# B&R Automation Studio project CleanChemi_SiteManagementSystem (part 24)

```iecst
		IF gSkid_LR[IdxSkids_LR].Alarms.ALARM_P203.11 AND gServices.Alarms.Internal.Alarms_State_LR[IdxSkids_LR].ALARM_P203.11 = FALSE THEN
			IF gSkid_LR[IdxSkids_LR].ErrorInfo.Text = '' THEN
				gSkid_LR[IdxSkids_LR].ErrorInfo.Text		:= 'ALARM_P203.11';
				gSkid_LR[IdxSkids_LR].ErrorInfo.State		:= 'Warning';
				gSkid_LR[IdxSkids_LR].ErrorInfo.Severity	:= 2;
				gSkid_LR[IdxSkids_LR].Error := TRUE;
				gServices.Alarms.Internal.Alarms_State_LR[IdxSkids_LR].ALARM_P203.11 := TRUE;
			END_IF
		END_IF;

		IF gSkid_LR[IdxSkids_LR].Alarms.ALARM_P203.12 AND gServices.Alarms.Internal.Alarms_State_LR[IdxSkids_LR].ALARM_P203.12 = FALSE THEN
			IF gSkid_LR[IdxSkids_LR].ErrorInfo.Text = '' THEN
				gSkid_LR[IdxSkids_LR].ErrorInfo.Text		:= 'ALARM_P203.12';
				gSkid_LR[IdxSkids_LR].ErrorInfo.State		:= 'Warning';
				gSkid_LR[IdxSkids_LR].ErrorInfo.Severity	:= 2;
				gSkid_LR[IdxSkids_LR].Error := TRUE;
				gServices.Alarms.Internal.Alarms_State_LR[IdxSkids_LR].ALARM_P203.12 := TRUE;
			END_IF
		END_IF;

		IF gSkid_LR[IdxSkids_LR].Alarms.ALARM_P203.13 AND gServices.Alarms.Internal.Alarms_State_LR[IdxSkids_LR].ALARM_P203.13 = FALSE THEN
			IF gSkid_LR[IdxSkids_LR].ErrorInfo.Text = '' THEN
				gSkid_LR[IdxSkids_LR].ErrorInfo.Text		:= 'ALARM_P203.13';
				gSkid_LR[IdxSkids_LR].ErrorInfo.State		:= 'Warning';
				gSkid_LR[IdxSkids_LR].ErrorInfo.Severity	:= 2;
				gSkid_LR[IdxSkids_LR].Error := TRUE;
				gServices.Alarms.Internal.Alarms_State_LR[IdxSkids_LR].ALARM_P203.13 := TRUE;
			END_IF
		END_IF;

		IF gSkid_LR[IdxSkids_LR].Alarms.ALARM_P203.14 AND gServices.Alarms.Internal.Alarms_State_LR[IdxSkids_LR].ALARM_P203.14 = FALSE THEN
			IF gSkid_LR[IdxSkids_LR].ErrorInfo.Text = '' THEN
				gSkid_LR[IdxSkids_LR].ErrorInfo.Text		:= 'ALARM_P203.14';
				gSkid_LR[IdxSkids_LR].ErrorInfo.State		:= 'Warning';
				gSkid_LR[IdxSkids_LR].ErrorInfo.Severity	:= 2;
				gSkid_LR[IdxSkids_LR].Error := TRUE;
				gServices.Alarms.Internal.Alarms_State_LR[IdxSkids_LR].ALARM_P203.14 := TRUE;
			END_IF
		END_IF;

		IF gSkid_LR[IdxSkids_LR].Alarms.ALARM_P203.15 AND gServices.Alarms.Internal.Alarms_State_LR[IdxSkids_LR].ALARM_P203.15 = FALSE THEN
			IF gSkid_LR[IdxSkids_LR].ErrorInfo.Text = '' THEN
				gSkid_LR[IdxSkids_LR].ErrorInfo.Text		:= 'ALARM_P203.15';
				gSkid_LR[IdxSkids_LR].ErrorInfo.State		:= 'Warning';
				gSkid_LR[IdxSkids_LR].ErrorInfo.Severity	:= 2;
				gSkid_LR[IdxSkids_LR].Error := TRUE;
				gServices.Alarms.Internal.Alarms_State_LR[IdxSkids_LR].ALARM_P203.15 := TRUE;
			END_IF
		END_IF;
	END_IF;

	(*********************************************************************Dont Touch This Code**********************************************************************)
	IF gSkid_LR[IdxSkids_LR].Error AND gSkid_LR[IdxSkids_LR].AlarmsInitialized AND gSkid_LR[IdxSkids_LR].Pmax_General_Variables.UNIT_ID <> 0 AND gUnit_LR[IdxSkids_LR] <> 0 THEN
		CASE gSkid_LR[IdxSkids_LR].ErrorInfo.Severity OF
			1:
				gSkid_LR[IdxSkids_LR].tempAlarm.name				:= UINT_TO_STRING(gUnit_LR[IdxSkids_LR]);
				gSkid_LR[IdxSkids_LR].tempAlarm.name				:= CONCAT('Skid',gSkid_LR[IdxSkids_LR].tempAlarm.name);
				gSkid_LR[IdxSkids_LR].tempAlarm.name				:= CONCAT(gSkid_LR[IdxSkids_LR].tempAlarm.name,'Severity1');
				gSkid_LR[IdxSkids_LR].tempAlarm.allowMultiple		:= TRUE;
				gSkid_LR[IdxSkids_LR].tempAlarm.addText[0]		:= gSkid_LR[IdxSkids_LR].ErrorInfo.State;
				gSkid_LR[IdxSkids_LR].tempAlarm.addText[1]		:= gSkid_LR[IdxSkids_LR].ErrorInfo.Text;

				HA_Array_AddTop(ADR(gServices.Alarms.In.AlarmList), SIZEOF(gServices.Alarms.In.AlarmList), ADR(gSkid_LR[IdxSkids_LR].tempAlarm), SIZEOF(gSkid_LR[IdxSkids_LR].tempAlarm));
			2:
				gSkid_LR[IdxSkids_LR].tempAlarm.name				:=  UINT_TO_STRING(gUnit_LR[IdxSkids_LR]);
				gSkid_LR[IdxSkids_LR].tempAlarm.name				:= CONCAT('Skid',gSkid_LR[IdxSkids_LR].tempAlarm.name);
				gSkid_LR[IdxSkids_LR].tempAlarm.name				:= CONCAT(gSkid_LR[IdxSkids_LR].tempAlarm.name,'Severity2');
				gSkid_LR[IdxSkids_LR].tempAlarm.allowMultiple		:= TRUE;
				gSkid_LR[IdxSkids_LR].tempAlarm.addText[0]		:= gSkid_LR[IdxSkids_LR].ErrorInfo.State;
				gSkid_LR[IdxSkids_LR].tempAlarm.addText[1]		:= gSkid_LR[IdxSkids_LR].ErrorInfo.Text;

				HA_Array_AddTop(ADR(gServices.Alarms.In.AlarmList), SIZEOF(gServices.Alarms.In.AlarmList), ADR(gSkid_LR[IdxSkids_LR].tempAlarm), SIZEOF(gSkid_LR[IdxSkids_LR].tempAlarm));
			3:
				gSkid_LR[IdxSkids_LR].tempAlarm.name				:=  UINT_TO_STRING(gUnit_LR[IdxSkids_LR]);
				gSkid_LR[IdxSkids_LR].tempAlarm.name				:= CONCAT('Skid',gSkid_LR[IdxSkids_LR].tempAlarm.name);
				gSkid_LR[IdxSkids_LR].tempAlarm.name				:= CONCAT(gSkid_LR[IdxSkids_LR].tempAlarm.name,'Severity3');
				gSkid_LR[IdxSkids_LR].tempAlarm.allowMultiple		:= TRUE;
				gSkid_LR[IdxSkids_LR].tempAlarm.addText[0]		:= gSkid_LR[IdxSkids_LR].ErrorInfo.State;
				gSkid_LR[IdxSkids_LR].tempAlarm.addText[1]		:= gSkid_LR[IdxSkids_LR].ErrorInfo.Text;

				HA_Array_AddTop(ADR(gServices.Alarms.In.AlarmList), SIZEOF(gServices.Alarms.In.AlarmList), ADR(gSkid_LR[IdxSkids_LR].tempAlarm), SIZEOF(gSkid_LR[IdxSkids_LR].tempAlarm));
			4:
				gSkid_LR[IdxSkids_LR].tempAlarm.name				:=  UINT_TO_STRING(gUnit_LR[IdxSkids_LR]);
				gSkid_LR[IdxSkids_LR].tempAlarm.name				:= CONCAT('Skid',gSkid_LR[IdxSkids_LR].tempAlarm.name);
				gSkid_LR[IdxSkids_LR].tempAlarm.name				:= CONCAT(gSkid_LR[IdxSkids_LR].tempAlarm.name,'Severity4');
				gSkid_LR[IdxSkids_LR].tempAlarm.allowMultiple		:= TRUE;
				gSkid_LR[IdxSkids_LR].tempAlarm.addText[0]		:= gSkid_LR[IdxSkids_LR].ErrorInfo.State;
				gSkid_LR[IdxSkids_LR].tempAlarm.addText[1]		:= gSkid_LR[IdxSkids_LR].ErrorInfo.Text;

				HA_Array_AddTop(ADR(gServices.Alarms.In.AlarmList), SIZEOF(gServices.Alarms.In.AlarmList), ADR(gSkid_LR[IdxSkids_LR].tempAlarm), SIZEOF(gSkid_LR[IdxSkids_LR].tempAlarm));
			5:

				gSkid_LR[IdxSkids_LR].tempAlarm.name				:=  UINT_TO_STRING(gUnit_LR[IdxSkids_LR]);
				gSkid_LR[IdxSkids_LR].tempAlarm.name				:= CONCAT('Skid',gSkid_LR[IdxSkids_LR].tempAlarm.name);
				gSkid_LR[IdxSkids_LR].tempAlarm.name				:= CONCAT(gSkid_LR[IdxSkids_LR].tempAlarm.name,'Severity5');
				gSkid_LR[IdxSkids_LR].tempAlarm.allowMultiple		:= TRUE;
				gSkid_LR[IdxSkids_LR].tempAlarm.addText[0]		:= gSkid_LR[IdxSkids_LR].ErrorInfo.State;
				gSkid_LR[IdxSkids_LR].tempAlarm.addText[1]		:= gSkid_LR[IdxSkids_LR].ErrorInfo.Text;

				HA_Array_AddTop(ADR(gServices.Alarms.In.AlarmList), SIZEOF(gServices.Alarms.In.AlarmList), ADR(gSkid_LR[IdxSkids_LR].tempAlarm), SIZEOF(gSkid_LR[IdxSkids_LR].tempAlarm));
		END_CASE

		gSkid_LR[IdxSkids_LR].Error := FALSE;

	END_IF

	brsmemset(ADR(gSkid_LR[IdxSkids_LR].ErrorInfo),0,SIZEOF(gSkid_LR[IdxSkids_LR].ErrorInfo));

	gServices.Alarms.Internal.MpAlarmXHistory_0.DeviceName 						:= ADR(gServices.DeviceName);

	//Set Unit Number and Add Alarms
	IF (gSkid_LR[IdxSkids_LR].Pmax_General_Variables.UNIT_ID <> 0 AND (gUnit_LR[IdxSkids_LR] <> gSkid_LR[IdxSkids_LR].Pmax_General_Variables.UNIT_ID))
		OR (gUnit_LR[IdxSkids_LR] <> 0 AND gVis.Alarms.Active.FilterString_LR[IdxSkids_LR] = '') THEN

		gUnit_LR[IdxSkids_LR] := gSkid_LR[IdxSkids_LR].Pmax_General_Variables.UNIT_ID;

		gSkid_LR[IdxSkids_LR].AlarmName	 := UINT_TO_STRING(gUnit_LR[IdxSkids_LR]);
		gSkid_LR[IdxSkids_LR].AlarmName	 := CONCAT('Skid',gSkid_LR[IdxSkids_LR].AlarmName	);

		gSkid_LR[IdxSkids_LR].i := 1;

		SkidNumberINT := UINT_TO_STRING(gUnit_LR[IdxSkids_LR]);

		gVis.Alarms.Active.FilterString_LR[IdxSkids_LR] := CONCAT('[{"value":',SkidNumberINT);
		gVis.Alarms.Active.FilterString_LR[IdxSkids_LR] :=  CONCAT(gVis.Alarms.Active.FilterString_LR[IdxSkids_LR] ,',"conditionType":"==","columnPosition":1}]');

	END_IF;

	// Case for handling the alarm history
	CASE gServices.Alarms.Internal.StateExportHistory OF
		0:
			IF gServices.Alarms.In.ExportHistory THEN
				HA_AlarmX_Helper(gAlarmXCore,'',HA_ALARMX_ACTION_LOG_ONLY,'HISTORY EXPORTED',FALSE);
				gServices.Alarms.In.ExportHistory 									:= FALSE;
				gServices.Alarms.Internal.MpAlarmXHistory_0.Export 				:= TRUE;
				gServices.Alarms.Internal.StateExportHistory 						:= 10;
			ELSIF gServices.Alarms.In.ClearHistory THEN
				HA_AlarmX_Helper(gAlarmXCore,'',HA_ALARMX_ACTION_LOG_ONLY,'HISTORY CLEARED',FALSE);
				gServices.Alarms.In.ClearHistory 									:= FALSE;
				MpAlarmXClearHistory(gAlarmXHistory);
			END_IF;
		10:
			IF gServices.Alarms.Internal.MpAlarmXHistory_0.CommandDone OR gServices.Alarms.Internal.MpAlarmXHistory_0.Error THEN
				gServices.Alarms.Internal.MpAlarmXHistory_0.Export 				:= FALSE;
				gServices.Alarms.Internal.StateExportHistory 						:= 0;
			END_IF;
	END_CASE;

	//	IF gMain.ErrorReset THEN
	//		gServices.Alarms.In.ResetAlarms 											:= TRUE;
	//	END_IF;

	// Case for handling the alarm resetting
	CASE gServices.Alarms.Internal.StateResetAlarms OF
		0:
			IF gServices.Alarms.In.ResetAlarms OR gVis.Global.ErrorReset THEN
				HA_AlarmX_Helper(gAlarmXCore,'',HA_ALARMX_ACTION_LOG_ONLY,'ACKNOWLEDGE ALL',FALSE);
				gServices.Alarms.In.ResetAlarms 									:= FALSE;
				gVis.Alarms.Active.UIConnect.AcknowledgeAll 							:= TRUE;
				gServices.Alarms.Internal.CTON_ResetDelay(IN := FALSE);
				gServices.Alarms.Internal.StateResetAlarms 						:= 10;
			END_IF;
		10:
			// give UI time to process the reset
			IF gServices.Alarms.Internal.CTON_ResetDelay.Q THEN
				gServices.Alarms.Internal.CTON_ResetDelay(IN := FALSE);
				gServices.Alarms.Internal.StateResetAlarms 						:= 0;
				gVis.Global.ErrorReset := FALSE;
			ELSE
				gServices.Alarms.Internal.CTON_ResetDelay(IN := TRUE, PT := T#250ms);
			END_IF;
	END_CASE;

	//Create Alarms
	CASE gSkid_LR[IdxSkids_LR].i OF
		0:
			//IDLE
		1:
			gSkid_LR[IdxSkids_LR].AlarmName	 := UINT_TO_STRING(gUnit_LR[IdxSkids_LR]);
			gSkid_LR[IdxSkids_LR].AlarmName	 := CONCAT('Skid',gSkid_LR[IdxSkids_LR].AlarmName	);
			HA_brsstrcat(ADR(gSkid_LR[IdxSkids_LR].AlarmName), ADR('Severity1'), SIZEOF(gSkid_LR[IdxSkids_LR].AlarmName));
			gSkid_LR[IdxSkids_LR].AlarmCfg.Message												:= '{$$IAT/Alarm.';
			HA_brsstrcat(ADR(gSkid_LR[IdxSkids_LR].AlarmCfg.Message), ADR('Severity1'), SIZEOF(gSkid_LR[IdxSkids_LR].AlarmCfg.Message));
			HA_brsstrcat(ADR(gSkid_LR[IdxSkids_LR].AlarmCfg.Message), ADR('}'), SIZEOF(gSkid_LR[IdxSkids_LR].AlarmCfg.Message));
			gSkid_LR[IdxSkids_LR].AlarmCfg.Code													:= gUnit_LR[IdxSkids_LR];
			gSkid_LR[IdxSkids_LR].AlarmCfg.Severity												:= 1;
			gSkid_LR[IdxSkids_LR].AlarmCfg.Behavior.AutoReset									:= TRUE;
			gSkid_LR[IdxSkids_LR].AlarmCfg.Behavior.Acknowledge 									:= mpALARMX_ACK_REQ;
			gSkid_LR[IdxSkids_LR].AlarmCfg.Behavior.MultipleInstances 							:= TRUE;
			gSkid_LR[IdxSkids_LR].AlarmCfg.Behavior.ReactionUntilAcknowledged					:= TRUE;
			gSkid_LR[IdxSkids_LR].AlarmCfg.Behavior.HistoryReport.AcknowledgedToUnacknowledged := FALSE;
			gSkid_LR[IdxSkids_LR].AlarmCfg.Behavior.HistoryReport.ActiveToInactive := FALSE;
			gSkid_LR[IdxSkids_LR].AlarmCfg.Behavior.HistoryReport.InactiveToActive := TRUE;
			gSkid_LR[IdxSkids_LR].AlarmCfg.Behavior.HistoryReport.Reactivation := FALSE;
			gSkid_LR[IdxSkids_LR].AlarmCfg.Behavior.HistoryReport.UnacknowledgedToAcknowledged := FALSE;
			gSkid_LR[IdxSkids_LR].MpAlarmXConfigAlarm.Save				:= TRUE;

		2:
			gSkid_LR[IdxSkids_LR].AlarmName	 := UINT_TO_STRING(gUnit_LR[IdxSkids_LR]);
			gSkid_LR[IdxSkids_LR].AlarmName	 := CONCAT('Skid',gSkid_LR[IdxSkids_LR].AlarmName	);
			HA_brsstrcat(ADR(gSkid_LR[IdxSkids_LR].AlarmName), ADR('Severity2'), SIZEOF(gSkid_LR[IdxSkids_LR].AlarmName));
			gSkid_LR[IdxSkids_LR].AlarmCfg.Message												:= '{$$IAT/Alarm.';
			HA_brsstrcat(ADR(gSkid_LR[IdxSkids_LR].AlarmCfg.Message), ADR('Severity2'), SIZEOF(gSkid_LR[IdxSkids_LR].AlarmCfg.Message));
			HA_brsstrcat(ADR(gSkid_LR[IdxSkids_LR].AlarmCfg.Message), ADR('}'), SIZEOF(gSkid_LR[IdxSkids_LR].AlarmCfg.Message));
			gSkid_LR[IdxSkids_LR].AlarmCfg.Code													:= gUnit_LR[IdxSkids_LR];
			gSkid_LR[IdxSkids_LR].AlarmCfg.Severity												:= 2;
			gSkid_LR[IdxSkids_LR].AlarmCfg.Behavior.AutoReset									:= TRUE;
			gSkid_LR[IdxSkids_LR].AlarmCfg.Behavior.Acknowledge 									:= mpALARMX_ACK_REQ;
			gSkid_LR[IdxSkids_LR].AlarmCfg.Behavior.MultipleInstances 							:= TRUE;
			gSkid_LR[IdxSkids_LR].AlarmCfg.Behavior.ReactionUntilAcknowledged					:= TRUE;
			gSkid_LR[IdxSkids_LR].AlarmCfg.Behavior.HistoryReport.AcknowledgedToUnacknowledged := FALSE;
			gSkid_LR[IdxSkids_LR].AlarmCfg.Behavior.HistoryReport.ActiveToInactive := FALSE;
			gSkid_LR[IdxSkids_LR].AlarmCfg.Behavior.HistoryReport.InactiveToActive := TRUE;
			gSkid_LR[IdxSkids_LR].AlarmCfg.Behavior.HistoryReport.Reactivation := FALSE;
			gSkid_LR[IdxSkids_LR].AlarmCfg.Behavior.HistoryReport.UnacknowledgedToAcknowledged := FALSE;
			gSkid_LR[IdxSkids_LR].MpAlarmXConfigAlarm.Save				:= TRUE;

		3:
			gSkid_LR[IdxSkids_LR].AlarmName	 := UINT_TO_STRING(gUnit_LR[IdxSkids_LR]);
			gSkid_LR[IdxSkids_LR].AlarmName	 := CONCAT('Skid',gSkid_LR[IdxSkids_LR].AlarmName	);
			HA_brsstrcat(ADR(gSkid_LR[IdxSkids_LR].AlarmName), ADR('Severity3'), SIZEOF(gSkid_LR[IdxSkids_LR].AlarmName));
			gSkid_LR[IdxSkids_LR].AlarmCfg.Message												:= '{$$IAT/Alarm.';
			HA_brsstrcat(ADR(gSkid_LR[IdxSkids_LR].AlarmCfg.Message), ADR('Severity3'), SIZEOF(gSkid_LR[IdxSkids_LR].AlarmCfg.Message));
			HA_brsstrcat(ADR(gSkid_LR[IdxSkids_LR].AlarmCfg.Message), ADR('}'), SIZEOF(gSkid_LR[IdxSkids_LR].AlarmCfg.Message));
			gSkid_LR[IdxSkids_LR].AlarmCfg.Code													:= gUnit_LR[IdxSkids_LR];
			gSkid_LR[IdxSkids_LR].AlarmCfg.Severity												:= 3;
			gSkid_LR[IdxSkids_LR].AlarmCfg.Behavior.AutoReset									:= TRUE;
			gSkid_LR[IdxSkids_LR].AlarmCfg.Behavior.Acknowledge 									:= mpALARMX_ACK_REQ;
			gSkid_LR[IdxSkids_LR].AlarmCfg.Behavior.MultipleInstances 							:= TRUE;
			gSkid_LR[IdxSkids_LR].AlarmCfg.Behavior.ReactionUntilAcknowledged					:= TRUE;
			gSkid_LR[IdxSkids_LR].AlarmCfg.Behavior.HistoryReport.AcknowledgedToUnacknowledged := FALSE;
			gSkid_LR[IdxSkids_LR].AlarmCfg.Behavior.HistoryReport.ActiveToInactive := FALSE;
			gSkid_LR[IdxSkids_LR].AlarmCfg.Behavior.HistoryReport.InactiveToActive := TRUE;
			gSkid_LR[IdxSkids_LR].AlarmCfg.Behavior.HistoryReport.Reactivation := FALSE;
			gSkid_LR[IdxSkids_LR].AlarmCfg.Behavior.HistoryReport.UnacknowledgedToAcknowledged := FALSE;
			gSkid_LR[IdxSkids_LR].MpAlarmXConfigAlarm.Save				:= TRUE;

		4:
			gSkid_LR[IdxSkids_LR].AlarmName	 := UINT_TO_STRING(gUnit_LR[IdxSkids_LR]);
			gSkid_LR[IdxSkids_LR].AlarmName	 := CONCAT('Skid',gSkid_LR[IdxSkids_LR].AlarmName	);
			HA_brsstrcat(ADR(gSkid_LR[IdxSkids_LR].AlarmName), ADR('Severity4'), SIZEOF(gSkid_LR[IdxSkids_LR].AlarmName));
			gSkid_LR[IdxSkids_LR].AlarmCfg.Message												:= '{$$IAT/Alarm.';
			HA_brsstrcat(ADR(gSkid_LR[IdxSkids_LR].AlarmCfg.Message), ADR('Severity4'), SIZEOF(gSkid_LR[IdxSkids_LR].AlarmCfg.Message));
			HA_brsstrcat(ADR(gSkid_LR[IdxSkids_LR].AlarmCfg.Message), ADR('}'), SIZEOF(gSkid_LR[IdxSkids_LR].AlarmCfg.Message));
			gSkid_LR[IdxSkids_LR].AlarmCfg.Code													:= gUnit_LR[IdxSkids_LR];
			gSkid_LR[IdxSkids_LR].AlarmCfg.Severity												:= 4;
			gSkid_LR[IdxSkids_LR].AlarmCfg.Behavior.AutoReset									:= TRUE;
			gSkid_LR[IdxSkids_LR].AlarmCfg.Behavior.Acknowledge 									:= mpALARMX_ACK_REQ;
			gSkid_LR[IdxSkids_LR].AlarmCfg.Behavior.MultipleInstances 							:= TRUE;
			gSkid_LR[IdxSkids_LR].AlarmCfg.Behavior.ReactionUntilAcknowledged					:= TRUE;
			gSkid_LR[IdxSkids_LR].AlarmCfg.Behavior.HistoryReport.AcknowledgedToUnacknowledged := FALSE;
			gSkid_LR[IdxSkids_LR].AlarmCfg.Behavior.HistoryReport.ActiveToInactive := FALSE;
			gSkid_LR[IdxSkids_LR].AlarmCfg.Behavior.HistoryReport.InactiveToActive := TRUE;
			gSkid_LR[IdxSkids_LR].AlarmCfg.Behavior.HistoryReport.Reactivation := FALSE;
			gSkid_LR[IdxSkids_LR].AlarmCfg.Behavior.HistoryReport.UnacknowledgedToAcknowledged := FALSE;
			gSkid_LR[IdxSkids_LR].MpAlarmXConfigAlarm.Save				:= TRUE;
		5:
			gSkid_LR[IdxSkids_LR].AlarmName	 := UINT_TO_STRING(gUnit_LR[IdxSkids_LR]);
			gSkid_LR[IdxSkids_LR].AlarmName	 := CONCAT('Skid',gSkid_LR[IdxSkids_LR].AlarmName	);
			HA_brsstrcat(ADR(gSkid_LR[IdxSkids_LR].AlarmName), ADR('Severity5'), SIZEOF(gSkid_LR[IdxSkids_LR].AlarmName));
			gSkid_LR[IdxSkids_LR].AlarmCfg.Message												:= '{$$IAT/Alarm.';
			HA_brsstrcat(ADR(gSkid_LR[IdxSkids_LR].AlarmCfg.Message), ADR('Severity5'), SIZEOF(gSkid_LR[IdxSkids_LR].AlarmCfg.Message));
			HA_brsstrcat(ADR(gSkid_LR[IdxSkids_LR].AlarmCfg.Message), ADR('}'), SIZEOF(gSkid_LR[IdxSkids_LR].AlarmCfg.Message));
			gSkid_LR[IdxSkids_LR].AlarmCfg.Code													:= gUnit_LR[IdxSkids_LR];
			gSkid_LR[IdxSkids_LR].AlarmCfg.Severity												:= 5;
			gSkid_LR[IdxSkids_LR].AlarmCfg.Behavior.AutoReset									:= TRUE;
			gSkid_LR[IdxSkids_LR].AlarmCfg.Behavior.Acknowledge 									:= mpALARMX_ACK_REQ;
			gSkid_LR[IdxSkids_LR].AlarmCfg.Behavior.MultipleInstances 							:= TRUE;
			gSkid_LR[IdxSkids_LR].AlarmCfg.Behavior.ReactionUntilAcknowledged					:= TRUE;
			gSkid_LR[IdxSkids_LR].AlarmCfg.Behavior.HistoryReport.AcknowledgedToUnacknowledged := FALSE;
			gSkid_LR[IdxSkids_LR].AlarmCfg.Behavior.HistoryReport.ActiveToInactive := FALSE;
			gSkid_LR[IdxSkids_LR].AlarmCfg.Behavior.HistoryReport.InactiveToActive := TRUE;
			gSkid_LR[IdxSkids_LR].AlarmCfg.Behavior.HistoryReport.Reactivation := FALSE;
			gSkid_LR[IdxSkids_LR].AlarmCfg.Behavior.HistoryReport.UnacknowledgedToAcknowledged := FALSE;
			gSkid_LR[IdxSkids_LR].MpAlarmXConfigAlarm.Save				:= TRUE;

		6:
			gSkid_LR[IdxSkids_LR].AlarmName	 := UINT_TO_STRING(gUnit_LR[IdxSkids_LR]);
			gSkid_LR[IdxSkids_LR].AlarmName	 := CONCAT('Skid',gSkid_LR[IdxSkids_LR].AlarmName	);
			HA_brsstrcat(ADR(gSkid_LR[IdxSkids_LR].AlarmName), ADR('CmdIgnored'), SIZEOF(gSkid_LR[IdxSkids_LR].AlarmName));
			gSkid_LR[IdxSkids_LR].AlarmCfg.Message												:= '{$$IAT/Alarm.';
			HA_brsstrcat(ADR(gSkid_LR[IdxSkids_LR].AlarmCfg.Message), ADR(gSkid_LR[IdxSkids_LR].AlarmName), SIZEOF(gSkid_LR[IdxSkids_LR].AlarmCfg.Message));
			HA_brsstrcat(ADR(gSkid_LR[IdxSkids_LR].AlarmCfg.Message), ADR('}'), SIZEOF(gSkid_LR[IdxSkids_LR].AlarmCfg.Message));
			gSkid_LR[IdxSkids_LR].AlarmCfg.Code													:= gUnit_LR[IdxSkids_LR] + 6;
			gSkid_LR[IdxSkids_LR].AlarmCfg.Severity												:= 0;
			gSkid_LR[IdxSkids_LR].AlarmCfg.Behavior.AutoReset									:= TRUE;
			gSkid_LR[IdxSkids_LR].AlarmCfg.Behavior.Acknowledge 									:= mpALARMX_ACK_REQ;
			gSkid_LR[IdxSkids_LR].AlarmCfg.Behavior.MultipleInstances 							:= TRUE;
			gSkid_LR[IdxSkids_LR].AlarmCfg.Behavior.ReactionUntilAcknowledged					:= TRUE;
			gSkid_LR[IdxSkids_LR].AlarmCfg.Behavior.HistoryReport.AcknowledgedToUnacknowledged := FALSE;
			gSkid_LR[IdxSkids_LR].AlarmCfg.Behavior.HistoryReport.ActiveToInactive := FALSE;
			gSkid_LR[IdxSkids_LR].AlarmCfg.Behavior.HistoryReport.InactiveToActive := TRUE;
			gSkid_LR[IdxSkids_LR].AlarmCfg.Behavior.HistoryReport.Reactivation := FALSE;
			gSkid_LR[IdxSkids_LR].AlarmCfg.Behavior.HistoryReport.UnacknowledgedToAcknowledged := FALSE;
			gSkid_LR[IdxSkids_LR].MpAlarmXConfigAlarm.Save				:= TRUE;
		7:
			gSkid_LR[IdxSkids_LR].AlarmStartupDelay.IN := TRUE;

			IF 	gSkid_LR[IdxSkids_LR].AlarmStartupDelay.Q THEN
				gSkid_LR[IdxSkids_LR].AlarmsInitialized := TRUE;
			END_IF;

	END_CASE

	gSkid_LR[IdxSkids_LR].AlarmStartupDelay(PT := T#30s);

	gSkid_LR[IdxSkids_LR].MpAlarmXConfigAlarm.MpLink			:= ADR(gAlarmXCore);
	gSkid_LR[IdxSkids_LR].MpAlarmXConfigAlarm.Enable			:= TRUE;
	gSkid_LR[IdxSkids_LR].MpAlarmXConfigAlarm.Name				:= ADR(gSkid_LR[IdxSkids_LR].AlarmName);
	gSkid_LR[IdxSkids_LR].MpAlarmXConfigAlarm.Configuration	:= ADR(gSkid_LR[IdxSkids_LR].AlarmCfg);

	IF gSkid_LR[IdxSkids_LR].MpAlarmXConfigAlarm.CommandDone THEN
		IF gSkid_LR[IdxSkids_LR].i < 7 THEN
			gSkid_LR[IdxSkids_LR].i := gSkid_LR[IdxSkids_LR].i + 1;
		ELSE
			//Do nothing
		END_IF;

		gSkid_LR[IdxSkids_LR].MpAlarmXConfigAlarm.Save := FALSE;
	END_IF;

	gSkid_LR[IdxSkids_LR].MpAlarmXConfigAlarm();

END_ACTION
```

- Visualisation Logical/mappView (not shown)

### Program Logical/Vis (IEC)

#### Main.st - Init, cyclic, exit code
```iecst
PROGRAM _INIT

	brsmemset(ADR(gVis.Main.Out.IPAddressDataProv_HR),0,SIZEOF(gVis.Main.Out.IPAddressDataProv_HR));
	brsmemset(ADR(gVis.Main.Out.IPAddressDataProv_LR),0,SIZEOF(gVis.Main.Out.IPAddressDataProv_LR));

	//Set IP Address for screen
	gVis.Main.Out.SkidIPAddress_LR := SLAVE_IP_ADDRESSES_LR;
	gVis.Main.Out.SkidIPAddress_HR := SLAVE_IP_ADDRESSES_HR;

END_PROGRAM

PROGRAM _CYCLIC

	//Grab Unit ID and Create Dropdown List
	FOR IdxSkids_LR := 0 TO MAX_SKIDS_LR DO

		IF gSkid_LR[IdxSkids_LR].Pmax_General_Variables.UNIT_ID = 0 THEN
			gVis.Main.Internal.IP_WSTRING_Temp := STRING_TO_WSTRING(SLAVE_IP_ADDRESSES_LR[IdxSkids_LR]);
			WString2DataProvider(ADR(gVis.Main.Internal.IP_WSTRING_Temp),IdxSkids_LR,ADR(gVis.Main.Out.IPAddressDataProv_LR[IdxSkids_LR]));
		ELSE
			gVis.Main.Internal.IP_WSTRING_Temp := UINT_TO_WSTRING(gSkid_LR[IdxSkids_LR].Pmax_General_Variables.UNIT_ID );
			WString2DataProvider(ADR(gVis.Main.Internal.IP_WSTRING_Temp),gSkid_LR[IdxSkids_LR].Pmax_General_Variables.UNIT_ID,ADR(gVis.Main.Out.IPAddressDataProv_LR[IdxSkids_LR]));
		END_IF;

	END_FOR

	FOR IdxSkids_HR := 0 TO MAX_SKIDS_HR DO

		IF gSkid_HR[IdxSkids_HR].Pmax_General_Variables.UNIT_ID = 0 THEN
			gVis.Main.Internal.IP_WSTRING_Temp := STRING_TO_WSTRING(SLAVE_IP_ADDRESSES_HR[IdxSkids_HR]);
			WString2DataProvider(ADR(gVis.Main.Internal.IP_WSTRING_Temp),IdxSkids_HR,ADR(gVis.Main.Out.IPAddressDataProv_HR[IdxSkids_HR]));
		ELSE
			gVis.Main.Internal.IP_WSTRING_Temp := UINT_TO_WSTRING(gSkid_HR[IdxSkids_HR].Pmax_General_Variables.UNIT_ID);
			WString2DataProvider(ADR(gVis.Main.Internal.IP_WSTRING_Temp),gSkid_HR[IdxSkids_HR].Pmax_General_Variables.UNIT_ID,ADR(gVis.Main.Out.IPAddressDataProv_HR[IdxSkids_HR]));
		END_IF;

	END_FOR

	//Main Page Widget Vis
	Vis_Main_HR;
	Vis_Main_LR;

	//Vis Action Calls
	Login_User_API;

	//Alarm Page Logic
	Alarms_Active;
	//	Alarms_History;

END_PROGRAM

PROGRAM _EXIT
	(* Insert code here *)

END_PROGRAM
```

#### Types.typ - Local data types
```iecst
TYPE
	USER_LOGIN_ENUM :
		(
		WAITING_FOR_LOGIN_I,
		LOGIN_USER_W,
		LOGIN_USER_C,
		LOGIN_SUCCESS,
		DELETE_USER_C,
		DELETE_USER_W,
		DELETE_USER_SUCCESS,
		DELETE_USER_ERROR,
		LOGIN_ERROR
		);
END_TYPE
```

#### Variables.var - Local variables
```iecst
VAR
	sampleTrigger : BOOL := FALSE;
	samplingTimer : TON := (0);
	bufferIndex : INT := 0;
	SkidNumberINT : STRING[5] := '';
	Idx_AlarmList : INT := 0;
	API_Login_FB_0 : API_Login_FB := (0);
	Header : httpRequestHeader_t := (0);
	CLIENT_LOGIN_STATE : USER_LOGIN_ENUM := WAITING_FOR_LOGIN_I;
	Client : httpsClient := (0);
	IdxClients_AlarmCheck : INT := 0;
	IdxClients : INT := 0;
	ArUserDelete_0 : ArUserDelete := (0);
	ArUserCreate_0 : ArUserCreate := (0);
	IdxSkids_HR : INT := 0;
	IdxSkids_LR : INT := 0;
	IndxNumber : USINT;
END_VAR
```

#### Alarms_Active.st
```iecst
ACTION Alarms_Active:

//	IF gVis.Alarms_Global.Active.Reset THEN
//		gVis.Alarms_Global.Active.Reset											:= FALSE;
//		gVis.Global.ErrorReset													:= TRUE;
//		brsmemset(ADR(gServices.Alarms_Global.Internal.Alarms_State),0,SIZEOF(gServices.Alarms_Global.Internal.Alarms_State));
//	END_IF;
//
	IF gVis.Alarms_Global.Active.PageUp THEN
		IF gVis.Alarms_Global.Active.SelectedIndex > 0 THEN
			gVis.Alarms_Global.Active.SelectedIndex := gVis.Alarms_Global.Active.SelectedIndex - 1;
		END_IF;
		gVis.Alarms_Global.Active.PageUp												:= FALSE;
	ELSIF gVis.Alarms_Global.Active.PageDown THEN
		gVis.Alarms_Global.Active.SelectedIndex := gVis.Alarms_Global.Active.SelectedIndex + 1;
		gVis.Alarms_Global.Active.PageDown												:= FALSE;
	END_IF;

	brsmemset(ADR(gVis.Alarms_Global.Active.TableConfig),0,SIZEOF(gVis.Alarms_Global.Active.TableConfig));
	HA_brsstrcat(ADR(gVis.Alarms_Global.Active.TableConfig),ADR('{"specRows": [ {"from":'),SIZEOF(gVis.Alarms_Global.Active.TableConfig));
	IF gVis.Alarms_Global.Active.UIConnect.AlarmList.MaxSelection = 0 THEN
		IF gVis.Alarms_Global.Active.UIConnect.AlarmList.Timestamp[0] = '' THEN
			gVis.Alarms_Global.Active.TempINT										:= 0;
		ELSE
			gVis.Alarms_Global.Active.TempINT										:= 1;
		END_IF;
	ELSE
		gVis.Alarms_Global.Active.TempINT											:= UINT_TO_INT(gVis.Alarms_Global.Active.UIConnect.AlarmList.MaxSelection)+1;
	END_IF;
	gVis.Alarms_Global.Active.TempSTRING 											:= INT_TO_STRING(gVis.Alarms_Global.Active.TempINT);
	HA_brsstrcat(ADR(gVis.Alarms_Global.Active.TableConfig),ADR(gVis.Alarms_Global.Active.TempSTRING),SIZEOF(gVis.Alarms_Global.Active.TableConfig));
	HA_brsstrcat(ADR(gVis.Alarms_Global.Active.TableConfig),ADR(', "to":'),SIZEOF(gVis.Alarms_Global.Active.TableConfig));
	gVis.Alarms_Global.Active.TempINT												:= 49;
	gVis.Alarms_Global.Active.TempSTRING 											:= INT_TO_STRING(gVis.Alarms_Global.Active.TempINT);
	HA_brsstrcat(ADR(gVis.Alarms_Global.Active.TableConfig),ADR(gVis.Alarms_Global.Active.TempSTRING),SIZEOF(gVis.Alarms_Global.Active.TableConfig));
	HA_brsstrcat(ADR(gVis.Alarms_Global.Active.TableConfig),ADR(', "visible":false} ]}'),SIZEOF(gVis.Alarms_Global.Active.TableConfig));

	//	IF gVis.Alarms_Global.Active.SelectedIndex <> gVis.Alarms_Global.Active.SelectedIndex_Temp THEN
	//
	//		FOR IdxSkids_HR := 0 TO MAX_SKIDS_HR DO
	//			IF gUnit_HR[IdxSkids_HR] = gVis.Alarms_HR.Active.UIConnect.AlarmList.Code[gVis.Alarms_HR.Active.SelectedIndex]  THEN
	//				gVis.Alarms_HR.Active.SelectedSkidIdx := IdxSkids_HR;
	//				EXIT;
	//			END_IF;
	//		END_FOR;
	//		gVis.Alarms_HR.Active.SelectedIndex_Temp := gVis.Alarms_HR.Active.SelectedIndex;
	//	END_IF;
	//
	//	IF gVis.Alarms_LR.Active.SelectedIndex <> gVis.Alarms_LR.Active.SelectedIndex_Temp THEN
	//		FOR IdxSkids_LR := 0 TO MAX_SKIDS DO
	//			IF gUnit_LR[IdxSkids_LR] = gVis.Alarms_LR.Active.UIConnect.AlarmList.Code[gVis.Alarms_LR.Active.SelectedIndex]  THEN
	//				gVis.Alarms_LR.Active.SelectedSkidIdx := IdxSkids_LR;
	//				EXIT;
	//			END_IF;
	//		END_FOR;
	//		gVis.Alarms_LR.Active.SelectedIndex_Temp := gVis.Alarms_LR.Active.SelectedIndex;
	//	END_IF;

	FOR IdxClients_AlarmCheck := 0 TO MAX_CLIENTS DO

		IF gVis.Global.ClientInfo[IdxClients_AlarmCheck].SelectedAlrmIndx <> gVis.Global.ClientInfo[IdxClients_AlarmCheck].SelectedAlrmIndx_Temp THEN
			gVis.Global.ClientInfo[IdxClients_AlarmCheck].SelectedAlrmIndx_Temp := gVis.Global.ClientInfo[IdxClients_AlarmCheck].SelectedAlrmIndx;
			FOR IdxSkids_LR := 0 TO MAX_SKIDS_LR DO
				IF gVis.Alarms_Global.Active.UIConnect.AlarmList.Code[gVis.Global.ClientInfo[IdxClients_AlarmCheck].SelectedAlrmIndx] = gUnit_LR[IdxSkids_LR] THEN
					gVis.Global.ClientInfo[IdxClients_AlarmCheck].SelectedAlrm_UnitID :=  UINT_TO_STRING(gUnit_LR[IdxSkids_LR]);
					gVis.Global.ClientInfo[IdxClients_AlarmCheck].SelectedAlrm_Skid := 'LR';

					EXIT;
				ELSIF IdxSkids_LR = MAX_SKIDS_LR THEN
					FOR IdxSkids_HR := 0 TO MAX_SKIDS_HR DO
						IF gVis.Alarms_Global.Active.UIConnect.AlarmList.Code[gVis.Global.ClientInfo[IdxClients_AlarmCheck].SelectedAlrmIndx] = gUnit_HR[IdxSkids_HR] THEN
							gVis.Global.ClientInfo[IdxClients_AlarmCheck].SelectedAlrm_UnitID := UINT_TO_STRING(gUnit_HR[IdxSkids_HR]);
							gVis.Global.ClientInfo[IdxClients_AlarmCheck].SelectedAlrm_Skid := 'HR';
							EXIT;
						END_IF;
					END_FOR
				END_IF
			END_FOR;
		END_IF;

	END_FOR;

	END_ACTION
```

#### Alarms_History.st
```iecst
ACTION Alarms_History:

	//gVis.Alarms.History.UIConnect.Language									:= gPar.System.LanguageCode;
	gVis.Alarms.History.UIConnect.AlarmList.SelectedIndex					:= gVis.Alarms.History.SelectedIndex;
	gVis.Alarms.History.UIConnect.AlarmList.PageUp							:= gVis.Alarms.History.PageUp;
	gVis.Alarms.History.PageUp												:= FALSE;
	gVis.Alarms.History.UIConnect.AlarmList.PageDown						:= gVis.Alarms.History.PageDown;
	gVis.Alarms.History.PageDown											:= FALSE;
	gServices.Alarms.In.ClearHistory									:= gVis.Alarms.History.Clear;
	gVis.Alarms.History.Clear												:= FALSE;
	gServices.Alarms.In.ExportHistory									:= gVis.Alarms.History.Export;
	gVis.Alarms.History.Export												:= FALSE;
	// Below loop sets the state variable to 1. Non 1 values are filtered from the table. This filters the history to only have when the alarm was triggered and not when it was acknowledged.
	FOR Idx_AlarmList := 0 TO 49 DO
		gVis.Alarms.History.State[Idx_AlarmList] 										:= 0;
		IF gVis.Alarms.History.UIConnect.AlarmList.NewState[Idx_AlarmList] = mpALARMX_STATE_ACTIVE THEN
			gVis.Alarms.History.State[Idx_AlarmList] 									:= 1;
		END_IF;
	END_FOR;

	brsmemset(ADR(gVis.Alarms.History.TableConfig),0,SIZEOF(gVis.Alarms.History.TableConfig));
	HA_brsstrcat(ADR(gVis.Alarms.History.TableConfig),ADR('{"specRows": [ {"from":'),SIZEOF(gVis.Alarms.History.TableConfig));
	IF gVis.Alarms.History.UIConnect.AlarmList.MaxSelection = 0 THEN
		IF gVis.Alarms.History.UIConnect.AlarmList.Timestamp[0] = '' THEN
			gVis.Alarms.History.TempINT										:= 0;
		ELSE
			gVis.Alarms.History.TempINT										:= 1;
		END_IF;
	ELSE
		gVis.Alarms.History.TempINT											:= UINT_TO_INT(gVis.Alarms.History.UIConnect.AlarmList.MaxSelection)+1;
	END_IF;
	gVis.Alarms.History.TempSTRING 											:= INT_TO_STRING(gVis.Alarms.History.TempINT);
	HA_brsstrcat(ADR(gVis.Alarms.History.TableConfig),ADR(gVis.Alarms.History.TempSTRING),SIZEOF(gVis.Alarms.History.TableConfig));
	HA_brsstrcat(ADR(gVis.Alarms.History.TableConfig),ADR(', "to":'),SIZEOF(gVis.Alarms.History.TableConfig));
	gVis.Alarms.History.TempINT												:= 49;
	gVis.Alarms.History.TempSTRING 											:= INT_TO_STRING(gVis.Alarms.History.TempINT);
	HA_brsstrcat(ADR(gVis.Alarms.History.TableConfig),ADR(gVis.Alarms.History.TempSTRING),SIZEOF(gVis.Alarms.History.TableConfig));
	HA_brsstrcat(ADR(gVis.Alarms.History.TableConfig),ADR(', "visible":false} ]}'),SIZEOF(gVis.Alarms.History.TableConfig));

END_ACTION
```

#### Login_User_API.st
```iecst
ACTION Login_User_API:

	Client.option 			:= httpOPTION_HTTP_11;
	Client.pHost 			:= ADR('cci-api-development-wjc4fopyua-uc.a.run.app');

	Header.protocol			:= 'HTTP/1.1';
	Header.host				:= 'cci-api-development-wjc4fopyua-uc.a.run.app';
	Header.contentType		:= 'application/json';
	Header.connection		:= 'keep-alive';
	Header.userLine[0].name	:= 'User-Agent';
	Header.userLine[0].value := 'SCADA';

	CASE CLIENT_LOGIN_STATE OF

		WAITING_FOR_LOGIN_I:

			API_Login_FB_0.bExecute := FALSE;
			ArUserDelete_0.Execute := FALSE;

			FOR IdxClients := 0 TO MAX_CLIENTS DO
				IF gVis.Global.ClientInfo[IdxClients].LogoutRequest THEN
					gVis.Global.ClientInfo[IdxClients].LogoutRequest := FALSE;
					IF gVis.Global.ClientInfo[IdxClients].LoginBypass OR gVis.Global.ClientInfo[IdxClients].UserID = 'Anonymous' THEN
						CLIENT_LOGIN_STATE := DELETE_USER_SUCCESS;
					ELSE
						CLIENT_LOGIN_STATE := DELETE_USER_C;
					END_IF;
					EXIT;
				ELSIF NOT gVis.Global.ClientInfo[IdxClients].IsValid AND gVis.Global.ClientInfo[IdxClients].UserID <> '' THEN
					IF gVis.Global.ClientInfo[IdxClients].UserID <> 'Anonymous' AND NOT gVis.Global.ClientInfo[IdxClients].LoginBypass AND NOT gVis.Global.ClientInfo[IdxClients].LogoutRequest THEN
						CLIENT_LOGIN_STATE := DELETE_USER_C;
					END_IF
					brsmemset(ADR(gVis.Global.ClientInfo[IdxClients]),0,SIZEOF(gVis.Global.ClientInfo[IdxClients]));
					EXIT;
				ELSIF gVis.Global.ClientInfo[IdxClients].LoginRequest THEN
					gVis.Global.ClientInfo[IdxClients].LoginRequest := FALSE;
					CLIENT_LOGIN_STATE := LOGIN_USER_C;
					EXIT;
				END_IF;
			END_FOR;

		LOGIN_USER_C:

			API_Login_FB_0.bExecute := TRUE;
			API_Login_FB_0.sUser := gVis.Global.ClientInfo[IdxClients].User;
			API_Login_FB_0.sPassword := gVis.Global.ClientInfo[IdxClients].Password;

			CLIENT_LOGIN_STATE := LOGIN_USER_W;

		LOGIN_USER_W:

			IF API_Login_FB_0.Done THEN

				CLIENT_LOGIN_STATE := LOGIN_SUCCESS;
			ELSIF API_Login_FB_0.Error THEN
				CLIENT_LOGIN_STATE := LOGIN_ERROR;
			END_IF;

		LOGIN_SUCCESS:

			gVis.Global.ClientInfo[IdxClients].LoginSuccess := TRUE;
			gVis.Global.ClientInfo[IdxClients].API_ID := API_Login_FB_0.ReturnedID;
			gVis.Global.ClientInfo[IdxClients].API_FIRST_NAME := API_Login_FB_0.ReturnedFirstName;
			gVis.Global.ClientInfo[IdxClients].API_LAST_NAME := API_Login_FB_0.ReturnedLastName;

			CLIENT_LOGIN_STATE := WAITING_FOR_LOGIN_I;

		LOGIN_ERROR:
			//Insert code for error popup
			gVis.Global.ClientInfo[IdxClients].LoginSuccess := FALSE;
			gVis.Global.ClientInfo[IdxClients].LoginFailed := TRUE;
			gVis.Global.ClientInfo[IdxClients].LoginErrorInfo := API_Login_FB_0.ErrorInfo;
			API_Login_FB_0.bExecute := FALSE;

			CLIENT_LOGIN_STATE := WAITING_FOR_LOGIN_I;
		DELETE_USER_C:

			ArUserDelete_0.Execute := TRUE;
			ArUserDelete_0.UserName := gVis.Global.ClientInfo[IdxClients].UserID;

			CLIENT_LOGIN_STATE := DELETE_USER_W;
		DELETE_USER_W:

			IF ArUserDelete_0.Done THEN
				CLIENT_LOGIN_STATE := DELETE_USER_SUCCESS;
			ELSIF ArUserDelete_0.Error THEN
				CLIENT_LOGIN_STATE := DELETE_USER_ERROR;
			END_IF;

		DELETE_USER_SUCCESS:
			gVis.Global.ClientInfo[IdxClients].LogoutSuccess := TRUE;
			CLIENT_LOGIN_STATE := WAITING_FOR_LOGIN_I;
		DELETE_USER_ERROR:
			//Insert code for error popup
			CLIENT_LOGIN_STATE := WAITING_FOR_LOGIN_I;

	END_CASE;

	API_Login_FB_0(HttpClientRef := Client, RequestHeader := Header);

	ArUserDelete_0();
	ArUserCreate_0();

				END_ACTION
```
